// TIA Portal V17 export
// export: Created 2024-03-30T11:15:00.09983Z, ExportSetting WithDefaults, DisplayName Totally Integrated Automation Portal, DisplayVersion V17, DisplayName TIA Portal Openness, DisplayVersion V17, DisplayName TIA Portal Version Control Interface, DisplayVersion V17, DisplayName STEP 7 Professional, DisplayVersion V17, DisplayName STEP 7 Safety, DisplayVersion V17, DisplayName WinCC Advanced, DisplayVersion V17
TYPE "typ_Broadcast"
// stored: IsFailsafeCompliant false
   STRUCT
      ldt_ts : LDT;
      di_hardwareId : DInt;
      di_hardwareModel : DInt;
      s_softwareName : String;
      di_softwareVersion : DInt;
      s_message : String;
   END_STRUCT;
END_TYPE
